// TIA Portal V20 export
VAR_GLOBAL   // PLC tag table "默认变量表"
   Clock_Byte AT %MB0 : Byte;
   Clock_10Hz AT %M0.0 : Bool;
   Clock_5Hz AT %M0.1 : Bool;
   "Clock_2.5Hz" AT %M0.2 : Bool;
   Clock_2Hz AT %M0.3 : Bool;
   "Clock_1.25Hz" AT %M0.4 : Bool;
   Clock_1Hz AT %M0.5 : Bool;
   "Clock_0.625Hz" AT %M0.6 : Bool;
   "Clock_0.5Hz" AT %M0.7 : Bool;
   System_Byte AT %MB1 : Byte;
   FirstScan AT %M1.0 : Bool;
   DiagStatusUpdate AT %M1.1 : Bool;
   AlwaysTRUE AT %M1.2 : Bool;
   AlwaysFALSE AT %M1.3 : Bool;
   PositioningAxis_1_Actor_Interface_AddressIn AT %I129.0 : "PD_TEL5_IN";
   PositioningAxis_1_Actor_Interface_AddressOut AT %Q132.0 : "PD_TEL5_OUT";
   滑台伺服S200_Actor_Interface_AddressIn AT %I260.0 : "PD_TEL105_IN";
   滑台伺服S200_Actor_Interface_AddressOut AT %Q260.0 : "PD_TEL105_OUT";
   RLO_1 AT %M100.0 : Bool;
   RLO_0 AT %M100.1 : Bool;
   FirstCycle AT %M100.2 : Bool;
   S120正限位 AT %I0.0 : Bool;
   s120负限位 AT %I0.1 : Bool;
   s120原点信号 AT %I0.2 : Bool;
   滑台伺服S200_Actor_Interface_TorqueDataAddressIn AT %I280.0 : "PD_TEL750_IN";
   滑台伺服S200_Actor_Interface_TorqueDataAddressOut AT %Q280.0 : "PD_TEL750_OUT";
   S200原点信号 AT %I0.3 : Bool;
   S200正限位 AT %I0.4 : Bool;
   S200负限位 AT %I0.5 : Bool;
   Tag_1 AT %M10.5 : Bool;
   Tag_2 AT %M10.6 : Bool;
END_VAR
VAR_GLOBAL CONSTANT   // user constants
   PN_DevDiag_MaxModules_UserConst : Int := 128;   // Maximale Anzahl der Module in einer ET-Station (z.B. ET200...); WICHTIG: um Zykluszeit und Speicherplatz zu optimieren mögl. kleinen Wert hier einstellen / Max number of modules, for optimization of scantime and memory space keep small / Max 数量 of modules, 给 optimization of scantime 和 内存 space keep small
   PN_DevDiag_MaxDevices_UserConst : Int := 255;   // Maximale Anzahl der PN-Devices; WICHTIG: um Zykluszeit und Speicherplatz zu optimieren mögl. kleinen Wert hier einstellen / Max number of PN-devices, for optimization of scantime and memory space keep small / Max 数量 of PN-devices, 给 optimization of scantime 和 内存 space keep small
   Type_HMI : Int := 101;   // SICAR HMI / HMI
   "Type_HMI+External" : Int := 102;   // SICAR HMI&Ext. / HMI&External / SICAR HMI&外部
   Type_External : Int := 103;   // SICAR Ext / External / SICAR 外部
   Type_OperatorPanel : Int := 105;   // SICAR OperatorPanel / OperatorPanel
   No_of_DataSets_Counter : Int := 8;   // Anzahl Datensätze Zähler / Number of data sets Counter / 数量 of 数据 sets 计数器
   No_of_DataSets_ShiftCounter : Int := 8;   // Anzahl Datensätze Schichtzähler / Number of data sets Shift Counter / 数量 of 数据 sets 工作轮班 计数器
   No_of_DataSets_CycleTimer : Int := 8;   // Anzahl Datensätze Taktzeiten / Number of data sets Cycle Timer / 数量 of 数据 sets 周期 记时器
   No_of_DataSets_LimitValues : Int := 8;   // Anzahl Datensätze Grenzwerte / Number of data sets Limit Value / 数量 of 数据 sets 限制 值
   No_Drives : Int := 2;   // Anzahl Antriebe / Number of drives / 数量 of 驱动
   No_UserOperation_screens : Int := 2;   // Anzahl Anwender Bedien-Bilder / Number of UserOperation screens / 数量 of UserOperation screens
   No_OperationMODE : Int := 5;   // Anzahl verwendeter Betriebsarten Breiche (max.: 12) / Number of used operation mode areas (max.: 12 ) / 数量 of used 运行 模式 areas (max.: 12 )
   No_HMI_PANEL : Int := 5;   // Anzahl verwendeter HMI/Panel (Max.: 40: 8 HMIs + 32 Panels) / Number of used HMI/Panel (Max.: 40: 8 HMIs + 32 Panels) / 数量 of used HMI/Panel (Max.: 40: 8 HMIs + 32 Panels)
   EQUIPMENTDATA_STEPHISTORYLENGTH : Int := 149;   // Equipment Data Step History Array Length / 设备 数据 步 历史 Array 长度
   EQUIPMENTDATA_ACTIVEALARMSLENGTH : Int := 9;   // Equipment Data Active Alarms Array Length / 设备 数据 现行 警报 Array 长度
   No_Reader : Int := 5;   // Anzahl Lesestellen / Number of reader / 数量 of 读码器
   No_Fixtures : Int := 2;
   No_Valves : Int := 4;
   No_PP : Int := 4;
   OpMode07_No_Robot : Int := 4;   // Anzahl Antriebe / Number of Robots
   No_ES : Int := 4;   // Anzahl Antriebe / Number of drives
   No_GS : Int := 1;   // Anzahl Antriebe / Number of drives
   No_LC : Int := 1;   // Anzahl Antriebe / Number of drives
   No_LS : Int := 1;   // Anzahl Antriebe / Number of drives
   Single_Input : Int := 1;
   OSSD_Input : Int := 5;
   OP_Sum : SInt := 2;   // 工位总数
   HMI_AXISCTRL_COUNT_AXES_UPPER_LIM : Int := 5;   // Upper limit for number of axes in HMI (maximum number - 1)
END_VAR
